KUKA KRL program: ps_stb_res_c1.src, ps_stb_res_c1.dat

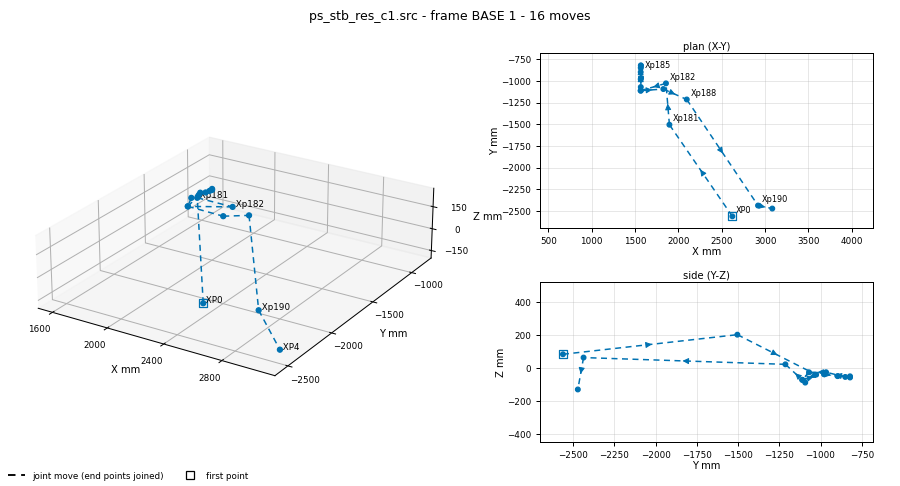
[picture p0: tool path of ps_stb_res_c1.src in frame BASE 1, 16 of 16 moves have a stored position in this frame; points joined in program order, loops and branches not executed]
--- ps_stb_res_c1.src ---
&ACCESS RVO
&REL 7
&COMMENT Solda GUN C1 respot
&PARAM DISKPATH = KRC:\R1\Program
DEF ps_stb_res_c1( )
;FOLD INI
;FOLD SPOTTECH INI
USERSPOT(#INIT)
;ENDFOLD (SPOTTECH INI)
;FOLD GRIPPERTECH INI
USER_GRP(0,DUMMY,DUMMY,GDEFAULT)
;ENDFOLD (GRIPPERTECH INI)
  ;FOLD USER INI
    ;Make your modifications here

  ;ENDFOLD (USER INI)
;ENDFOLD (INI)

; Caracterização dos meios de produção:
; Versão Atual:
; 08/06/2013 12:00 Name: P13.050-R1 CHANGES: Solda respot STB
; Gun C1 (F2 6640 0018 984)

chk_w2_wechs_ok ( )              ; CHECK C1

if MaxStandMenge (1) then
 MaxStandmengeErreicht (1)
endif

IF (NOT(GHOST())) THEN
if Elektrodenwechsel (1) then
 e_fraes2 ()
endif
ENDIF

;FOLD PTP P0 CONT Vel=100 % P_OLP20 Tool[2]:GUN C1 Base[1]:Actros;%{PE}%R 8.2.20,%MKUKATPBASIS,%CMOVE,%VPTP,%P 1:PTP, 2:P0, 3:C_DIS, 5:100, 7:P_OLP20
$BWDSTART=FALSE
PDAT_ACT=PP_OLP20
FDAT_ACT=FP0
BAS(#PTP_PARAMS,100)
PTP XP0 C_DIS
;ENDFOLD

;FOLD OUT 3334 'R1 solicita lib. soldar respot' State=TRUE ;%{PE}%R 8.2.20,%MKUKATPBASIS,%COUT,%VOUTX,%P 2:3334, 3:R1 solicita lib. soldar respot, 5:TRUE, 6:
$OUT[3334]=TRUE
;ENDFOLD
;FOLD WAIT FOR ( IN 3334 'Aguarda lib. Soldar respot' );%{PE}%R 8.2.20,%MKUKATPBASIS,%CEXT_WAIT_FOR,%VEXT_WAIT_FOR,%P 2:, 4:, 5:$IN, 6:3334, 7:Aguarda lib. Soldar respot, 9:
WAIT FOR  ( $IN[3334] )
;ENDFOLD
;FOLD OUT 3334 'R1 solicita lib. soldar respot' State=FALSE ;%{PE}%R 8.2.20,%MKUKATPBASIS,%COUT,%VOUTX,%P 2:3334, 3:R1 solicita lib. soldar respot, 5:FALSE, 6:
$OUT[3334]=FALSE
;ENDFOLD
;FOLD OUT 3348 'Fora area GEOBOX' State=FALSE ;%{PE}%R 8.2.20,%MKUKATPBASIS,%COUT,%VOUTX,%P 2:3348, 3:Fora area GEOBOX, 5:FALSE, 6:
$OUT[3348]=FALSE
;ENDFOLD

;FOLD PTP p181 CONT Vel=100 % P_OLP6 Tool[2]:GUN C1 Base[1]:Actros;%{PE}%R8.2,%MKUKATPBASIS,%CMOVE,%VPTP,%P 1:PTP, 2:p181, 3:C_DIS, 5:100, 7:P_OLP6
$BWDSTART = FALSE
PDAT_ACT= PP_OLP6
FDAT_ACT= Fp181
BAS(#PTP_PARAMS,100)
PTP Xp181 C_DIS
;ENDFOLD
;FOLD PTP p182 CONT Vel=100 % P_OLP7 Tool[2]:GUN C1 Base[1]:Actros;%{PE}%R8.2,%MKUKATPBASIS,%CMOVE,%VPTP,%P 1:PTP, 2:p182, 3:C_DIS, 5:100, 7:P_OLP7
$BWDSTART = FALSE
PDAT_ACT= PP_OLP7
FDAT_ACT= Fp182
BAS(#PTP_PARAMS,100)
PTP Xp182 C_DIS
;ENDFOLD
;FOLD PTP p183 CONT Vel=50 % P_OLP8 Tool[2]:GUN C1 Base[1]:Actros;%{PE}%R 8.2.20,%MKUKATPBASIS,%CMOVE,%VPTP,%P 1:PTP, 2:p183, 3:C_DIS, 5:50, 7:P_OLP8
$BWDSTART=FALSE
PDAT_ACT=PP_OLP8
FDAT_ACT=Fp183
BAS(#PTP_PARAMS,50)
PTP Xp183 C_DIS
;ENDFOLD
;FOLD PTP p184 CONT Vel=50 % P_OLP9 Tool[2]:GUN C1 Base[1]:Actros;%{PE}%R 8.2.20,%MKUKATPBASIS,%CMOVE,%VPTP,%P 1:PTP, 2:p184, 3:C_DIS, 5:50, 7:P_OLP9
$BWDSTART=FALSE
PDAT_ACT=PP_OLP9
FDAT_ACT=Fp184
BAS(#PTP_PARAMS,50)
PTP Xp184 C_DIS
;ENDFOLD
;FOLD PTP p185 CONT Vel=50 % P_OLP10 Tool[2]:GUN C1 Base[1]:Actros;%{PE}%R 8.2.20,%MKUKATPBASIS,%CMOVE,%VPTP,%P 1:PTP, 2:p185, 3:C_DIS, 5:50, 7:P_OLP10
$BWDSTART=FALSE
PDAT_ACT=PP_OLP10
FDAT_ACT=Fp185
BAS(#PTP_PARAMS,50)
PTP Xp185 C_DIS
;ENDFOLD

;FOLD PTP P2 Vel=50 % PDAT2 Tool[2]:GUN C1 Base[1]:Actros;%{PE}%R 8.2.20,%MKUKATPBASIS,%CMOVE,%VPTP,%P 1:PTP, 2:P2, 3:, 5:50, 7:PDAT2
$BWDSTART=FALSE
PDAT_ACT=PPDAT2
FDAT_ACT=FP2
BAS(#PTP_PARAMS,50)
PTP XP2
;ENDFOLD
;FOLD ; swp_60_4359;%{PE}%R 8.2.20,%MKUKATPBASIS,%CCOMMENT,%VNORMAL,%P 2:swp_60_4359
;ENDFOLD
;FOLD PTP swp_60_4359 P_OLP11 SPOT Gun=1 RETR CLS PgNo1=49 ACTIVE=1 Tool[2]:GUN C1 Base[1]:Actros;%{PE}%R 8.2.2,%MKUKATPSPOT,%CSPOT,%VPTP,%P 1:PTP, 2:swp_60_4359, 3:, 5:100, 7:P_OLP11, 10:1, 12:#FIRST, 14:#CLO, 16:49, 18:1, 20:1, 22:0, 24:1, 25:S_OLP1
$BWDSTART=FALSE
PDAT_ACT=PP_OLP11
FDAT_ACT=Fswp_60_4359
BAS(#PTP_PARAMS,PP_OLP11.VEL)
S_ACT.GUN=1
S_ACT.PAIR=SDEFAULT.PAIR
S_ACT.RETR=#CLO
S_ACT.CLO_TM=1
S_ACT.PGNO1=49
S_ACT.PGNO2=SDEFAULT.PGNO2
S_ACT.PRESS1=SDEFAULT.PRESS1
S_ACT.PRESS2=SDEFAULT.PRESS2
S_READY=FALSE
PTP Xswp_60_4359
USERSPOT(#SPOT, S_ACT)
WAIT FOR S_READY
;ENDFOLD

;FOLD ; swp_60_4363;%{PE}%R 8.2.20,%MKUKATPBASIS,%CCOMMENT,%VNORMAL,%P 2:swp_60_4363
;ENDFOLD
;FOLD PTP swp_60_4363 P_OLP12 SPOT Gun=1 RETR CLS PgNo1=50 ACTIVE=1 Tool[2]:GUN C1 Base[1]:Actros;%{PE}%R 8.2.2,%MKUKATPSPOT,%CSPOT,%VPTP,%P 1:PTP, 2:swp_60_4363, 3:, 5:100, 7:P_OLP12, 10:1, 12:#FIRST, 14:#CLO, 16:50, 18:1, 20:1, 22:0, 24:1, 25:S_OLP2
$BWDSTART=FALSE
PDAT_ACT=PP_OLP12
FDAT_ACT=Fswp_60_4363
BAS(#PTP_PARAMS,PP_OLP12.VEL)
S_ACT.GUN=1
S_ACT.PAIR=SDEFAULT.PAIR
S_ACT.RETR=#CLO
S_ACT.CLO_TM=1
S_ACT.PGNO1=50
S_ACT.PGNO2=SDEFAULT.PGNO2
S_ACT.PRESS1=SDEFAULT.PRESS1
S_ACT.PRESS2=SDEFAULT.PRESS2
S_READY=FALSE
PTP Xswp_60_4363
USERSPOT(#SPOT, S_ACT)
WAIT FOR S_READY
;ENDFOLD

;FOLD ; swp_60_4367;%{PE}%R 8.2.20,%MKUKATPBASIS,%CCOMMENT,%VNORMAL,%P 2:swp_60_4367
;ENDFOLD
;FOLD PTP swp_60_4367 P_OLP13 SPOT Gun=1 RETR CLS PgNo1=51 ACTIVE=1 Tool[2]:GUN C1 Base[1]:Actros;%{PE}%R 8.2.2,%MKUKATPSPOT,%CSPOT,%VPTP,%P 1:PTP, 2:swp_60_4367, 3:, 5:100, 7:P_OLP13, 10:1, 12:#FIRST, 14:#CLO, 16:51, 18:1, 20:1, 22:0, 24:1, 25:S_OLP3
$BWDSTART=FALSE
PDAT_ACT=PP_OLP13
FDAT_ACT=Fswp_60_4367
BAS(#PTP_PARAMS,PP_OLP13.VEL)
S_ACT.GUN=1
S_ACT.PAIR=SDEFAULT.PAIR
S_ACT.RETR=#CLO
S_ACT.CLO_TM=1
S_ACT.PGNO1=51
S_ACT.PGNO2=SDEFAULT.PGNO2
S_ACT.PRESS1=SDEFAULT.PRESS1
S_ACT.PRESS2=SDEFAULT.PRESS2
S_READY=FALSE
PTP Xswp_60_4367
USERSPOT(#SPOT, S_ACT)
WAIT FOR S_READY
;ENDFOLD

;FOLD ; swp_60_4373;%{PE}%R 8.2.20,%MKUKATPBASIS,%CCOMMENT,%VNORMAL,%P 2:swp_60_4373
;ENDFOLD
;FOLD PTP swp_60_4373 P_OLP14 SPOT Gun=1 RETR CLS PgNo1=52 ACTIVE=1 Tool[2]:GUN C1 Base[1]:Actros;%{PE}%R 8.2.2,%MKUKATPSPOT,%CSPOT,%VPTP,%P 1:PTP, 2:swp_60_4373, 3:, 5:100, 7:P_OLP14, 10:1, 12:#FIRST, 14:#CLO, 16:52, 18:1, 20:1, 22:0, 24:1, 25:S_OLP4
$BWDSTART=FALSE
PDAT_ACT=PP_OLP14
FDAT_ACT=Fswp_60_4373
BAS(#PTP_PARAMS,PP_OLP14.VEL)
S_ACT.GUN=1
S_ACT.PAIR=SDEFAULT.PAIR
S_ACT.RETR=#CLO
S_ACT.CLO_TM=1
S_ACT.PGNO1=52
S_ACT.PGNO2=SDEFAULT.PGNO2
S_ACT.PRESS1=SDEFAULT.PRESS1
S_ACT.PRESS2=SDEFAULT.PRESS2
S_READY=FALSE
PTP Xswp_60_4373
USERSPOT(#SPOT, S_ACT)
WAIT FOR S_READY
;ENDFOLD

;FOLD PTP p186 CONT Vel=80 % P_OLP15 Tool[2]:GUN C1 Base[1]:Actros;%{PE}%R 8.2.20,%MKUKATPBASIS,%CMOVE,%VPTP,%P 1:PTP, 2:p186, 3:C_DIS, 5:80, 7:P_OLP15
$BWDSTART=FALSE
PDAT_ACT=PP_OLP15
FDAT_ACT=Fp186
BAS(#PTP_PARAMS,80)
PTP Xp186 C_DIS
;ENDFOLD
;FOLD PTP p187 CONT Vel=100 % P_OLP16 Tool[2]:GUN C1 Base[1]:Actros;%{PE}%R8.2,%MKUKATPBASIS,%CMOVE,%VPTP,%P 1:PTP, 2:p187, 3:C_DIS, 5:100, 7:P_OLP16
$BWDSTART = FALSE
PDAT_ACT= PP_OLP16
FDAT_ACT= Fp187
BAS(#PTP_PARAMS,100)
PTP Xp187 C_DIS
;ENDFOLD
;FOLD PTP p188 CONT Vel=100 % P_OLP17 Tool[2]:GUN C1 Base[1]:Actros;%{PE}%R8.2,%MKUKATPBASIS,%CMOVE,%VPTP,%P 1:PTP, 2:p188, 3:C_DIS, 5:100, 7:P_OLP17
$BWDSTART = FALSE
PDAT_ACT= PP_OLP17
FDAT_ACT= Fp188
BAS(#PTP_PARAMS,100)
PTP Xp188 C_DIS
;ENDFOLD
;FOLD PTP p190 CONT Vel=100 % P_OLP19 Tool[2]:GUN C1 Base[1]:Actros;%{PE}%R8.2,%MKUKATPBASIS,%CMOVE,%VPTP,%P 1:PTP, 2:p190, 3:C_DIS, 5:100, 7:P_OLP19
$BWDSTART = FALSE
PDAT_ACT= PP_OLP19
FDAT_ACT= Fp190
BAS(#PTP_PARAMS,100)
PTP Xp190 C_DIS
;ENDFOLD
;FOLD PTP P4 CONT Vel=100 % PDAT4 Tool[2]:GUN C1 Base[1]:Actros;%{PE}%R 8.2.20,%MKUKATPBASIS,%CMOVE,%VPTP,%P 1:PTP, 2:P4, 3:C_DIS, 5:100, 7:PDAT4
$BWDSTART=FALSE
PDAT_ACT=PPDAT4
FDAT_ACT=FP4
BAS(#PTP_PARAMS,100)
PTP XP4 C_DIS
;ENDFOLD

;FOLD OUT 3348 'Fora area GEOBOX' State=TRUE ;%{PE}%R 8.2.20,%MKUKATPBASIS,%COUT,%VOUTX,%P 2:3348, 3:Fora area GEOBOX, 5:TRUE, 6:
$OUT[3348]=TRUE
;ENDFOLD

IF (NOT(GHOST())) THEN
if FraesAnf (1) then
 f_fraes2 ()
endif
ENDIF

END

--- ps_stb_res_c1.dat ---
&ACCESS RVO
&REL 7
&COMMENT Solda GUN C1 respot
&PARAM DISKPATH = KRC:\R1\Program
DEFDAT  ps_stb_res_c1
;FOLD EXTERNAL DECLARATIONS;%{PE}%MKUKATPBASIS,%CEXT,%VCOMMON,%P
;FOLD GRIPPERTECH EXT
EXT  H50 (INT  :IN,INT  :IN,INT  :IN,GRP_TYP  :IN )
;ENDFOLD (GRIPPERTECH EXT)
;FOLD SPOTTECH EXT
EXT  USERSPOT (S_COMMAND  :IN,SPOT_TYPE  :IN )
;ENDFOLD (SPOTTECH EXT)
;FOLD BASISTECH EXT;%{PE}%MKUKATPBASIS,%CEXT,%VEXT,%P
EXT  BAS (BAS_COMMAND  :IN,REAL  :IN )
DECL INT SUCCESS
;ENDFOLD (BASISTECH EXT)
;FOLD USER EXT;%{E}%MKUKATPUSER,%CEXT,%VEXT,%P
;Make your modifications here

;ENDFOLD (USER EXT)
;ENDFOLD (EXTERNAL DECLARATIONS)

;# ============ START PATH : swp_p13050r1_stb_res_c1 =============
DECL FDAT Fp181={TOOL_NO 2,BASE_NO 1,IPO_FRAME #BASE,POINT2[] " "}
DECL PDAT PP_OLP6={VEL 100.0,ACC 100.0,APO_DIST 100.0,APO_MODE #CDIS}
DECL E6POS Xp181={X 1896.36694,Y -1504.00305,Z 202.587402,A 140.237305,B -43.7405205,C 42.2965088,S 2,T 42,E1 -4648.65479,E2 0.0,E3 0.0,E4 0.0,E5 0.0,E6 0.0}
DECL FDAT Fp182={TOOL_NO 2,BASE_NO 1,IPO_FRAME #BASE,POINT2[] " "}
DECL PDAT PP_OLP7={VEL 100.0,ACC 100.0,APO_DIST 100.0,APO_MODE #CDIS}
DECL E6POS Xp182={X 1856.44495,Y -1026.70203,Z -39.5777397,A 106.560097,B -51.0617294,C 67.0245209,S 2,T 42,E1 -4823.9502,E2 0.0,E3 0.0,E4 0.0,E5 0.0,E6 0.0}
DECL FDAT Fp183={TOOL_NO 2,BASE_NO 1,IPO_FRAME #BASE,POINT2[] " "}
DECL PDAT PP_OLP8={VEL 100.0,ACC 100.0,APO_DIST 100.0,APO_MODE #CDIS}
DECL E6POS Xp183={X 1565.25696,Y -1110.33704,Z -71.3700027,A 90.0,B -38.0041008,C 90.0,S 2,T 42,E1 -5004.70117,E2 0.0,E3 0.0,E4 0.0,E5 0.0,E6 0.0}
DECL FDAT Fp184={TOOL_NO 2,BASE_NO 1,IPO_FRAME #BASE,POINT2[] " "}
DECL PDAT PP_OLP9={VEL 100.0,ACC 100.0,APO_DIST 100.0,APO_MODE #CDIS}
DECL E6POS Xp184={X 1565.24902,Y -978.995117,Z -37.5031319,A 90.0,B -21.7397594,C 90.0,S 2,T 42,E1 -5004.70117,E2 0.0,E3 0.0,E4 0.0,E5 0.0,E6 0.0}
DECL FDAT Fp185={TOOL_NO 2,BASE_NO 1,IPO_FRAME #BASE,POINT2[] " ",TQ_STATE FALSE}
DECL PDAT PP_OLP10={VEL 100.0,ACC 100.0,APO_DIST 100.0,APO_MODE #CDIS}
DECL E6POS Xp185={X 1565.25,Y -896.96698,Z -48.5442505,A 90.0772781,B -8.50728607,C 89.8862991,S 2,T 42,E1 -5004.70215,E2 0.0,E3 0.0,E4 0.0,E5 0.0,E6 0.0}
DECL FDAT Fswp_60_4359={TOOL_NO 2,BASE_NO 1,IPO_FRAME #BASE,POINT2[] " ",TQ_STATE FALSE}
DECL PDAT PP_OLP11={VEL 50.0,ACC 100.0,APO_DIST 0.0}
DECL SPOT_TYPE SS_OLP1={GUN 1,PAIR #FIRST,RETR #CLO,CLO_TM 0,PGNO1 1,PRESS1 1.0,PGNO2 0,PRESS2 0.0}
DECL E6POS Xswp_60_4359={X 1566.81604,Y -821.049194,Z -56.9380112,A 89.9963837,B -5.66864204,C 89.0004501,S 2,T 42,E1 -5004.70215,E2 0.0,E3 0.0,E4 0.0,E5 0.0,E6 0.0}
DECL FDAT Fswp_60_4363={TOOL_NO 2,BASE_NO 1,IPO_FRAME #BASE,POINT2[] " "}
DECL PDAT PP_OLP12={VEL 50.0,ACC 100.0,APO_DIST 0.0}
DECL SPOT_TYPE SS_OLP2={GUN 1,PAIR #FIRST,RETR #CLO,CLO_TM 0,PGNO1 1,PRESS1 1.0,PGNO2 0,PRESS2 0.0}
DECL E6POS Xswp_60_4363={X 1565.99902,Y -850.022217,Z -53.5922203,A 90.1103287,B -6.57939816,C 88.7786331,S 2,T 42,E1 -5004.70215,E2 0.0,E3 0.0,E4 0.0,E5 0.0,E6 0.0}
DECL FDAT Fswp_60_4367={TOOL_NO 2,BASE_NO 1,IPO_FRAME #BASE,POINT2[] " "}
DECL PDAT PP_OLP13={VEL 100.0,ACC 100.0,APO_DIST 0.0}
DECL SPOT_TYPE SS_OLP3={GUN 1,PAIR #FIRST,RETR #CLO,CLO_TM 0,PGNO1 1,PRESS1 1.0,PGNO2 0,PRESS2 0.0}
DECL E6POS Xswp_60_4367={X 1568.36206,Y -966.42749,Z -25.0264492,A 89.9996719,B -23.9013405,C 90.0008011,S 2,T 42,E1 -5004.70215,E2 0.0,E3 0.0,E4 0.0,E5 0.0,E6 0.0}
DECL FDAT Fswp_60_4373={TOOL_NO 2,BASE_NO 1,IPO_FRAME #BASE,POINT2[] " "}
DECL PDAT PP_OLP14={VEL 50.0,ACC 100.0,APO_DIST 0.0}
DECL SPOT_TYPE SS_OLP4={GUN 1,PAIR #FIRST,RETR #CLO,CLO_TM 0,PGNO1 1,PRESS1 1.0,PGNO2 0,PRESS2 0.0}
DECL E6POS Xswp_60_4373={X 1566.172,Y -1069.56897,Z -25.5048294,A 90.0002365,B -38.0078888,C 89.9996338,S 2,T 42,E1 -5004.70215,E2 0.0,E3 0.0,E4 0.0,E5 0.0,E6 0.0}
DECL FDAT Fp186={TOOL_NO 2,BASE_NO 1,IPO_FRAME #BASE,POINT2[] " "}
DECL PDAT PP_OLP15={VEL 100.0,ACC 100.0,APO_DIST 100.0,APO_MODE #CDIS}
DECL E6POS Xp186={X 1565.25806,Y -1110.96802,Z -70.6638107,A 90.0,B -45.8351402,C 90.0,S 2,T 42,E1 -5004.70117,E2 0.0,E3 0.0,E4 0.0,E5 0.0,E6 0.0}
DECL FDAT Fp187={TOOL_NO 2,BASE_NO 1,IPO_FRAME #BASE,POINT2[] " "}
DECL PDAT PP_OLP16={VEL 100.0,ACC 100.0,APO_DIST 100.0,APO_MODE #CDIS}
DECL E6POS Xp187={X 1826.30396,Y -1092.56799,Z -87.8626328,A 111.357002,B -59.1372108,C 62.2247314,S 2,T 42,E1 -5004.70117,E2 0.0,E3 0.0,E4 0.0,E5 0.0,E6 0.0}
DECL FDAT Fp188={TOOL_NO 2,BASE_NO 1,IPO_FRAME #BASE,POINT2[] " "}
DECL PDAT PP_OLP17={VEL 100.0,ACC 100.0,APO_DIST 100.0,APO_MODE #CDIS}
DECL E6POS Xp188={X 2096.43604,Y -1212.85095,Z 22.8050995,A 171.705002,B -47.6958504,C -2.87318301,S 2,T 42,E1 -4933.86914,E2 0.0,E3 0.0,E4 0.0,E5 0.0,E6 0.0}
DECL FDAT Fp190={TOOL_NO 2,BASE_NO 1,IPO_FRAME #BASE,POINT2[] " "}
DECL PDAT PP_OLP19={VEL 100.0,ACC 100.0,APO_DIST 100.0,APO_MODE #CDIS}
DECL E6POS Xp190={X 2918.8999,Y -2436.36304,Z 63.8172493,A -39.2407799,B 27.4611092,C -15.6265202,S 2,T 42,E1 -3436.99512,E2 0.0,E3 0.0,E4 0.0,E5 0.0,E6 0.0}
DECL BASIS_SUGG_T LAST_BASIS={POINT1[] "P4                      ",POINT2[] "P4                      ",CP_PARAMS[] "CPDAT0                  ",PTP_PARAMS[] "PDAT4                   ",CONT[] "C_DIS                   ",CP_VEL[] "2.0                     ",PTP_VEL[] "100                     ",SYNC_PARAMS[] "SYNCDAT                 ",SPL_NAME[] "S0                      "}
DECL SPOT_SUGG_T LAST_SPOT={GUN[] " 1                      ",RETR_CMD[] "#OPN                    ",CHOISE[] "#FIRST                  ",CLO_TM[] "0                       ",PGNO1[] " 1                      ",PRESS1[] "0                       ",PGNO2[] " 1                      ",PRESS2[] "0                       ",SPOT_PARAMS[] "NORMAL                  "}
DECL PDAT PP_OLP20={VEL 100.0,ACC 100.0,APO_DIST 100.0,APO_MODE #CDIS}
DECL E6POS XP0={X 2622.56494,Y -2561.18408,Z 83.8666992,A -129.9785,B -15.34513,C -14.8367596,S 2,T 42,E1 -3810.29102,E2 0.0,E3 0.0,E4 0.0,E5 0.0,E6 0.0}
DECL FDAT FP0={TOOL_NO 2,BASE_NO 1,IPO_FRAME #BASE,POINT2[] " ",TQ_STATE FALSE}
DECL E6POS XP2={X 1567.14197,Y -821.074585,Z -49.7357407,A 89.8357315,B -7.99154615,C 88.6038971,S 2,T 42,E1 -5004.70508,E2 0.0,E3 0.0,E4 0.0,E5 0.0,E6 0.0}
DECL FDAT FP2={TOOL_NO 2,BASE_NO 1,IPO_FRAME #BASE,POINT2[] " ",TQ_STATE FALSE}
DECL PDAT PPDAT2={VEL 100.0,ACC 100.0,APO_DIST 100.0,APO_MODE #CDIS}
DECL E6POS XP4={X 3083.12598,Y -2471.14209,Z -129.498703,A -5.38643312,B 6.33558083,C 0.0589020811,S 2,T 10,E1 -3852.87012,E2 0.0,E3 0.0,E4 0.0,E5 0.0,E6 0.0}
DECL FDAT FP4={TOOL_NO 2,BASE_NO 1,IPO_FRAME #BASE,POINT2[] " ",TQ_STATE FALSE}
DECL PDAT PPDAT4={VEL 100.0,ACC 100.0,APO_DIST 100.0,APO_MODE #CDIS}
ENDDAT
